(* IEC 61131-3 sources: SigmatekTestframework/src/Class/CStandardTestReport, 1 file *)

(* ---- CStandardTestReport.st ---- *)
(*!
<Class
	Name               = "CStandardTestReport"
	Revision           = "1.0"
	RealtimeTask       = "false"
	CyclicTask         = "false"
	BackgroundTask     = "false"
	Sigmatek           = "false"
	OSInterface        = "false"
	HighPriority       = "false"
	Automatic          = "false"
	UpdateMode         = "Prescan"
	SharedCommandTable = "true"
	Objectsize         = "(510,120)">
	<Channels>
	</Channels>
	<Network Name="CStandardTestReport">
		<!-- List of Components in this network -->
		<Components>
			<Object
				Name       = "_base"
				Class      = "CTestReportBase"
				Position   = "(218,120)"
				Visualized = "false">
				<Channels>
					<Server Name="Registered"/>
					<Client Name="clib"/>
					<Client Name="File"/>
					<Client Name="System"/>
				</Channels>
			</Object>
		</Components>
		<Comments>
		</Comments>
		<!-- List of Connections in this network -->
		<Connections>
			<Connection Source="this.Registered" Destination="_base.Registered" Vertices="(690,210),(518,210),"/>
		</Connections>
		<!-- Headerfiles -->
		<Options>
		</Options>
	</Network>
</Class>
*)
#pragma using CTestReportBase

CStandardTestReport : CLASS
: CTestReportBase
  //Servers:
  //Clients:
  //Variables:
  //Functions:

	FUNCTION VIRTUAL BuildFile
		VAR_OUTPUT
			eRetcode 	: ERetCode_t;
		END_VAR;

	FUNCTION VIRTUAL getFileName
		VAR_INPUT
			pFileName 	: ^CHAR;
			pFilePath 	: ^CHAR;
		END_VAR
		VAR_OUTPUT
			eRetcode 	: ERetCode_t;
		END_VAR;
  //Tables:
	FUNCTION @STD
		VAR_OUTPUT
			ret_code	: CONFSTATES;
		END_VAR;
	FUNCTION GLOBAL TAB @CT_;
END_CLASS;

//Exclude-SccX
(*
 **********************************************************************
 * \file CStandardTestReport.st
 *
 * Creates a simple Textfile as report
 *
 * Copyright (c) 2016,Hoox.Software, Helmbrechts
 * All Rights Reserved.
 *
 * Created on: 01.06.2016
 *     Author: dressel
 *
 **********************************************************************
 *)

//*********************************************************************
//
//
//
//
//*********************************************************************
FUNCTION VIRTUAL CStandardTestReport::getFileName
	VAR_INPUT
		pFileName 	: ^CHAR;
		pFilePath 	: ^CHAR;
	END_VAR
	VAR_OUTPUT
		eRetcode 	: ERetCode_t;
	END_VAR

   _strcpy(dest:= pFilePath, src:= "C:\Testrun");
   _strcpy(dest:= pFileName, src:= "Testlog1.txt");

   eRetcode := eDone;

END_FUNCTION

//*********************************************************************
//
//
//
//
//*********************************************************************
FUNCTION VIRTUAL CStandardTestReport::BuildFile
VAR_OUTPUT
   eRetcode 	: ERetCode_t;
END_VAR

   clearBuffer();

   addString(pData:= "Testreport");

   writeBuffer();

   addString(pData:= "___________________________________________" );

   writeBuffer();

   addString(pData:="Number of Suites: ");

   addValue(m_pTestLib^.NbSuites$DINT);

   writeBuffer();

   addString(pData:="Number of Tests: ");

   addValue(m_pTestLib^.NbRun$DINT);

   writeBuffer();

   addString(pData:="Number of Passed: ");

   addValue(m_pTestLib^.NbPassed$DINT);

   writeBuffer();

   addString(pData:="Number of Failed: ");

   addValue(m_pTestLib^.NbFailed$DINT);

   writeBuffer();

   addString(pData:= "___________________________________________" );

   writeBuffer();

   eRetcode := eDone;

END_FUNCTION
